PROGRAM MAIN
VAR
	m : INT;
END_VAR

m := m + 1;
PrgMqttCom();

END_PROGRAM

(* stored: Version 1.1.0.1, ProductVersion 3.1.4021.12
   POU MAIN: Id {db9963b7-0480-4e4a-a239-3a25f7a8c759}, SpecialFunc None *)
